{attribute 'GeneratedUsingTerminal: EL6201-0000-0017'}
{attribute addProperty BoxType "EL6201-0000-0017"}
{attribute addProperty Id "Slave_24A_DO0BOOL1Slave_24A_DO1BOOL1Slave_24A_DO2BOOL1Slave_24A_DO3BOOL1Slave_24B_DO0BOOL1Slave_24B_DO1BOOL1Slave_24B_DO2BOOL1Slave_24B_DO3BOOL1"}
{attribute addProperty CRC "3670023772"}
{attribute addProperty Size "8"}
TYPE Slave_24_Outputs_DAC01E5C :
STRUCT
	{attribute addProperty Name "Slave_24A_DO0"}
	Slave_24A_DO0 : BOOL;
	{attribute addProperty Name "Slave_24A_DO1"}
	Slave_24A_DO1 : BOOL;
	{attribute addProperty Name "Slave_24A_DO2"}
	Slave_24A_DO2 : BOOL;
	{attribute addProperty Name "Slave_24A_DO3"}
	Slave_24A_DO3 : BOOL;
	{attribute addProperty Name "Slave_24B_DO0"}
	Slave_24B_DO0 : BOOL;
	{attribute addProperty Name "Slave_24B_DO1"}
	Slave_24B_DO1 : BOOL;
	{attribute addProperty Name "Slave_24B_DO2"}
	Slave_24B_DO2 : BOOL;
	{attribute addProperty Name "Slave_24B_DO3"}
	Slave_24B_DO3 : BOOL;
END_STRUCT
END_TYPE

(* stored: Version 1.2.0.0, ProductVersion 3.1.4024.9
   DUT Slave_24_Outputs_DAC01E5C: Id {6e2e9fd5-d12a-4dab-aa06-5a20200f494a} *)
